// TIA Portal V16 export
// export: Created 2021-03-04T22:04:01.8053121Z, ExportSetting WithDefaults, DisplayName Totally Integrated Automation Portal, DisplayVersion V16, DisplayName TIA Portal Version Control Interface, DisplayVersion V16, DisplayName TIA Portal Openness, DisplayVersion V16, DisplayName SINAMICS Startdrive Advanced, DisplayVersion V16, DisplayName SINAMICS Startdrive G130, G150, S120, S150, SINAMICS MV, S210, DisplayVersion V16, DisplayName SINAMICS Startdrive G110M, G120, G120C, G120D, G120P, DisplayVersion V16, DisplayName STEP 7 Professional, DisplayVersion V16, DisplayName STEP 7 Safety, DisplayVersion V16, DisplayName WinCC Professional, DisplayVersion V16
FUNCTION_BLOCK "fbRoomCO2Control"   // FB13, LAD
{ S7_Optimized_Access := 'TRUE' }
VERSION : 0.1
// stored: AutoNumber true, IsIECCheckEnabled false, IsRetainMemResEnabled false, MemoryReserve 100, SetENOAutomatically false, UDAEnableTagReadback false
   VAR_INPUT
      iInCO2ReadingRaw { ExternalAccessible := 'False'; ExternalVisible := 'False'; ExternalWritable := 'False'} : Int;
   END_VAR
   VAR_OUTPUT
      bOutSolenoid { ExternalAccessible := 'False'; ExternalVisible := 'False'; ExternalWritable := 'False'} : Bool;
   END_VAR
   VAR
      AI_CO2Sensor { ExternalVisible := 'False'} : "fbAlarmedSetpoint";
   END_VAR
   VAR RETAIN
      Controls { ExternalVisible := 'False'} : Struct
         iModeCommand { ExternalVisible := 'False'} : Int;   // 0: Off, 1: Periodic Dosing
         tMeasurementInterval { ExternalVisible := 'False'} : Time := T#30s;   // Time between measurements
         tDosingDuration { ExternalVisible := 'False'} : Time := T#5s;   // Time to open solenoid if measurement is below setpoint
      END_STRUCT;
   END_VAR
   VAR
      Status { ExternalVisible := 'False'; ExternalWritable := 'False'} : Struct
         tElapsedMeasurement { ExternalVisible := 'False'; ExternalWritable := 'False'} : Time;
         tElapsedDosing { ExternalVisible := 'False'; ExternalWritable := 'False'} : Time;
      END_STRUCT;
   END_VAR
   VAR RETAIN
      TON_MeasurementCycle { ExternalAccessible := 'False'; ExternalVisible := 'False'; ExternalWritable := 'False'} : TON_TIME;
      TP_Dosing { ExternalAccessible := 'False'; ExternalVisible := 'False'; ExternalWritable := 'False'} : TP_TIME;
   END_VAR
   VAR_TEMP
      bCheckMeasurement : Bool;
   END_VAR
   VAR CONSTANT
      eMode_Off : Int := 0;   // forced off
      eMode_PeriodicDosing : Int := 2;   // auto
   END_VAR
   // AI_CO2Sensor.arrSetpoints[1].rSetpoint := 400.0;
   // AI_CO2Sensor.Config.rHighCalibration := 10000.0;
BEGIN

REGION Network 1 (SCL)
   // process CO2 sensor input
   #AI_CO2Sensor(#iInCO2ReadingRaw);

   // if mode is set to periodic dosing, run timer to periodically check value
   #bCheckMeasurement := #TON_MeasurementCycle.Q;
   #TON_MeasurementCycle(IN := #Controls.iModeCommand = #eMode_PeriodicDosing AND NOT #bCheckMeasurement,
                         PT := #Controls.tMeasurementInterval,
                         ET => #Status.tElapsedMeasurement);

   //if value is below setpoint, open valve for set duration
   #TP_Dosing(IN := #bCheckMeasurement AND #AI_CO2Sensor.rActual < #AI_CO2Sensor.rSetpoint,
               PT := #Controls.tDosingDuration,
               Q => #bOutSolenoid,
               ET => #Status.tElapsedDosing);
END_REGION
END_FUNCTION_BLOCK
